{attribute 'Tc2GvlVarNames'}
VAR_GLOBAL CONSTANT
	(* System_SHZ_Zustand_Status *)
	E_System_SHZ_Zustand_Status_Idle_Sperre					: SINT := 0;
	E_System_SHZ_Zustand_Status_Betriebsbereit				: SINT := 1;
	E_System_SHZ_Zustand_Status_Nachl_Pumpe					: SINT := 2;
	E_System_SHZ_Zustand_Status_Vorl_Pumpe					: SINT := 3;
	E_System_SHZ_Zustand_Status_Nachl_Regelventil			: SINT := 4;
	E_System_SHZ_Zustand_Status_Vorl_Regelventil			: SINT := 5;
	E_System_SHZ_Zustand_Status_Betrieb						: SINT := 6;
	E_System_SHZ_Zustand_Status_Betrieb_Sperre				: SINT := 7;
	E_System_SHZ_Zustand_Status_Stoerung					: SINT := 99;

	(* System_SHZ_Zustand_Regelung_Modus *)
	E_System_SHZ_Regelung_Modus_Automatik					: SINT := 0;
	E_System_SHZ_Regelung_Modus_Heizen_konst				: SINT := 1;
	E_System_SHZ_Regelung_Modus_Heizen_Kurve				: SINT := 2;
	E_System_SHZ_Regelung_Modus_Heizen_Kurve_Nachtabs		: SINT := 3;
	E_System_SHZ_Regelung_Modus_Kuehlen_konst				: SINT := -1;
	E_System_SHZ_Regelung_Modus_Kuehlen_Kurve				: SINT := -2;

END_VAR

(* stored: Version 1.1.0.1, ProductVersion 3.1.4024.9
   GVL Con_SHZ: Id {0883dfe4-1581-44ca-85ae-b4d5b91a6df6} *)
